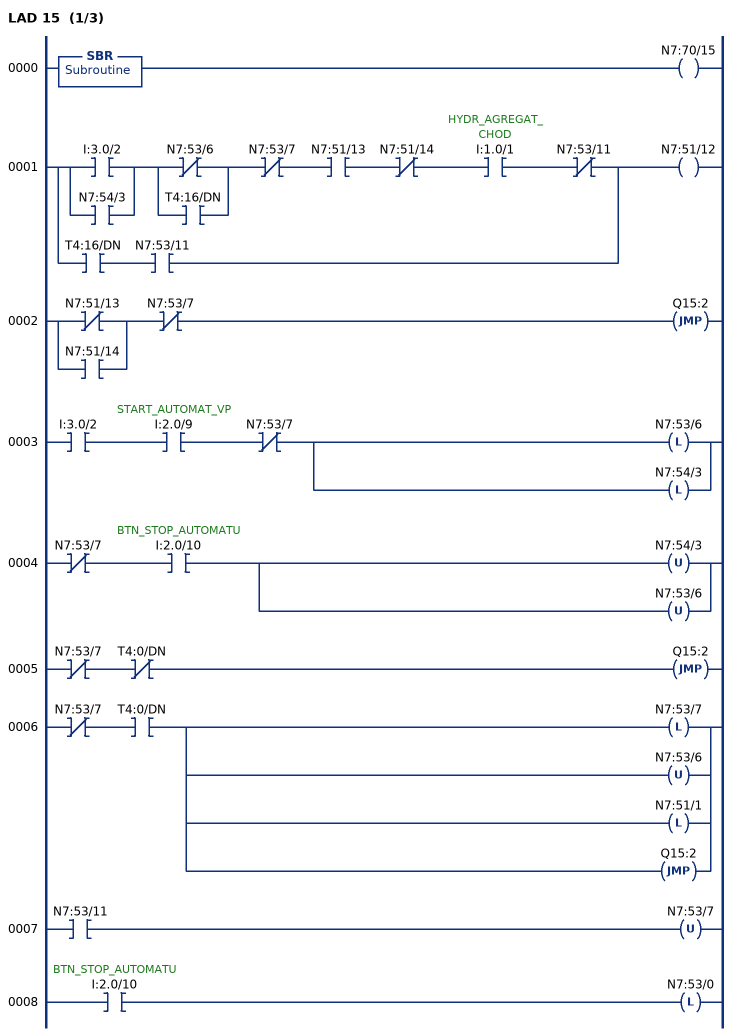
% Rung: 0 %
SOR SBR OTE N7:70/15 EOR
% Rung: 1 %
SOR BST BST XIC I:3.0/2 NXB XIC N7:54/3 BND BST XIO N7:53/6 NXB XIC T4:16/DN BND XIO N7:53/7 XIC N7:51/13 XIO N7:51/14 XIC I:1.0/1 XIO N7:53/11 NXB XIC T4:16/DN XIC N7:53/11 BND OTE N7:51/12 EOR
%   I:1.0/1  HYDR_AGREGAT_CHOD %
% Rung: 2 %
SOR BST XIO N7:51/13 NXB XIC N7:51/14 BND XIO N7:53/7 JMP Q15:2 EOR
% Rung: 3 %
SOR XIC I:3.0/2 XIC I:2.0/9 XIO N7:53/7 BST OTL N7:53/6 NXB OTL N7:54/3 BND EOR
%   I:2.0/9  START_AUTOMAT_VP %
% Rung: 4 %
SOR XIO N7:53/7 XIC I:2.0/10 BST OTU N7:54/3 NXB OTU N7:53/6 BND EOR
%   I:2.0/10  BTN_STOP_AUTOMATU %
% Rung: 5 %
SOR XIO N7:53/7 XIO T4:0/DN JMP Q15:2 EOR
% Rung: 6 %
SOR XIO N7:53/7 XIC T4:0/DN BST OTL N7:53/7 NXB OTU N7:53/6 NXB OTL N7:51/1 NXB JMP Q15:2 BND EOR
% Rung: 7 %
SOR XIC N7:53/11 OTU N7:53/7 EOR
% Rung: 8 %
SOR XIC I:2.0/10 OTL N7:53/0 EOR
%   I:2.0/10  BTN_STOP_AUTOMATU %

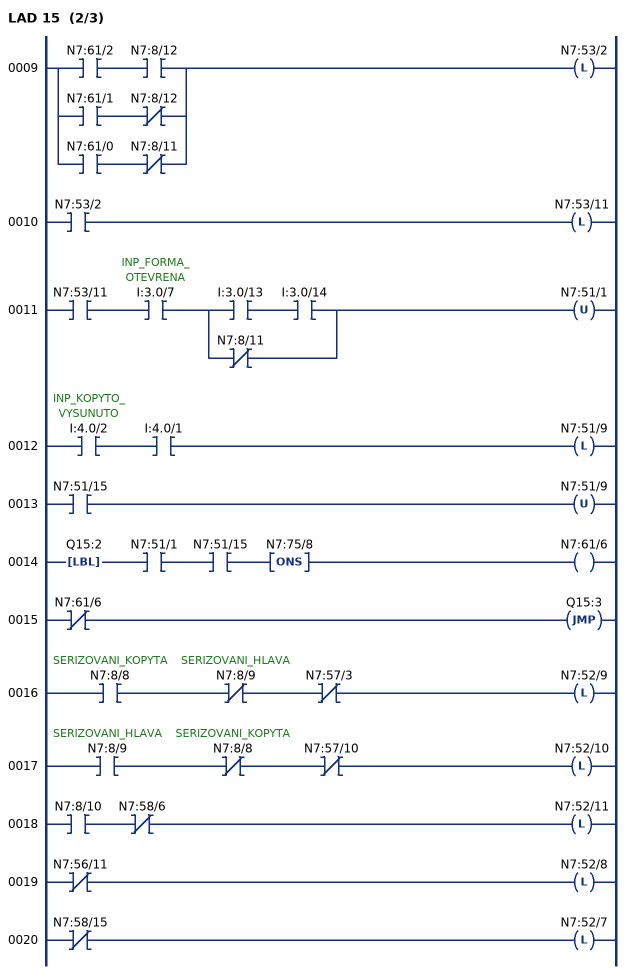
% Rung: 9 %
SOR BST XIC N7:61/2 XIC N7:8/12 NXB XIC N7:61/1 XIO N7:8/12 NXB XIC N7:61/0 XIO N7:8/11 BND OTL N7:53/2 EOR
% Rung: 10 %
SOR XIC N7:53/2 OTL N7:53/11 EOR
% Rung: 11 %
SOR XIC N7:53/11 XIC I:3.0/7 BST XIC I:3.0/13 XIC I:3.0/14 NXB XIO N7:8/11 BND OTU N7:51/1 EOR
%   I:3.0/7  INP_FORMA_OTEVRENA %
% Rung: 12 %
SOR XIC I:4.0/2 XIC I:4.0/1 OTL N7:51/9 EOR
%   I:4.0/2  INP_KOPYTO_VYSUNUTO %
% Rung: 13 %
SOR XIC N7:51/15 OTU N7:51/9 EOR
% Rung: 14 %
SOR LBL Q15:2 XIC N7:51/1 XIC N7:51/15 OSR N7:75/8 OTE N7:61/6 EOR
% Rung: 15 %
SOR XIO N7:61/6 JMP Q15:3 EOR
% Rung: 16 %
SOR XIC N7:8/8 XIO N7:8/9 XIO N7:57/3 OTL N7:52/9 EOR
%   N7:8/8  SERIZOVANI_KOPYTA %
%   N7:8/9  SERIZOVANI_HLAVA %
% Rung: 17 %
SOR XIC N7:8/9 XIO N7:8/8 XIO N7:57/10 OTL N7:52/10 EOR
%   N7:8/9  SERIZOVANI_HLAVA %
%   N7:8/8  SERIZOVANI_KOPYTA %
% Rung: 18 %
SOR XIC N7:8/10 XIO N7:58/6 OTL N7:52/11 EOR
% Rung: 19 %
SOR XIO N7:56/11 OTL N7:52/8 EOR
% Rung: 20 %
SOR XIO N7:58/15 OTL N7:52/7 EOR

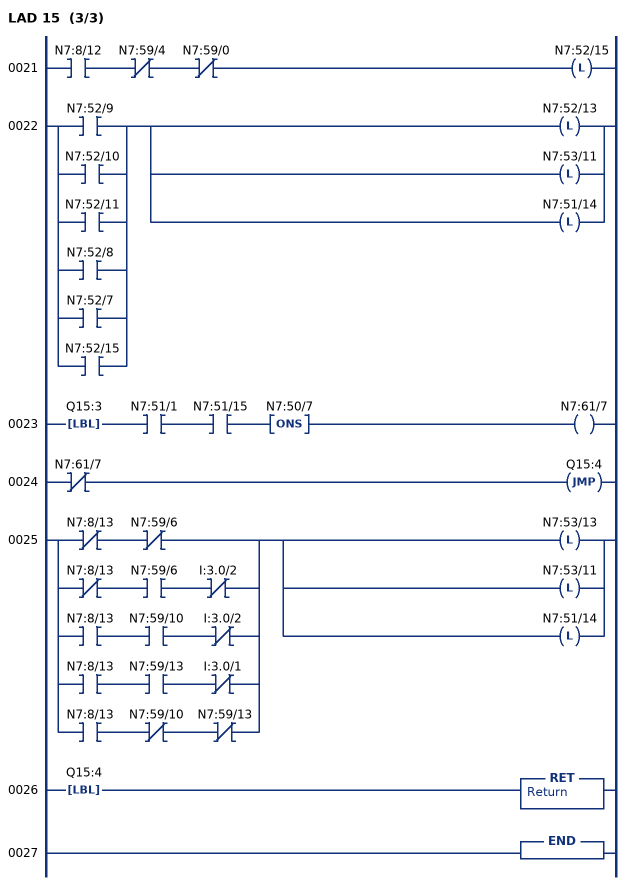
% Rung: 21 %
SOR XIC N7:8/12 XIO N7:59/4 XIO N7:59/0 OTL N7:52/15 EOR
% Rung: 22 %
SOR BST XIC N7:52/9 NXB XIC N7:52/10 NXB XIC N7:52/11 NXB XIC N7:52/8 NXB XIC N7:52/7 NXB XIC N7:52/15 BND BST OTL N7:52/13 NXB OTL N7:53/11 NXB OTL N7:51/14 BND EOR
% Rung: 23 %
SOR LBL Q15:3 XIC N7:51/1 XIC N7:51/15 OSR N7:50/7 OTE N7:61/7 EOR
% Rung: 24 %
SOR XIO N7:61/7 JMP Q15:4 EOR
% Rung: 25 %
SOR BST XIO N7:8/13 XIO N7:59/6 NXB XIO N7:8/13 XIC N7:59/6 XIO I:3.0/2 NXB XIC N7:8/13 XIC N7:59/10 XIO I:3.0/2 NXB XIC N7:8/13 XIC N7:59/13 XIO I:3.0/1 NXB XIC N7:8/13 XIO N7:59/10 XIO N7:59/13 BND BST OTL N7:53/13 NXB OTL N7:53/11 NXB OTL N7:51/14 BND EOR
% Rung: 26 %
SOR LBL Q15:4 RET EOR
% Rung: 27 %
SOR END EOR

LADDER 16
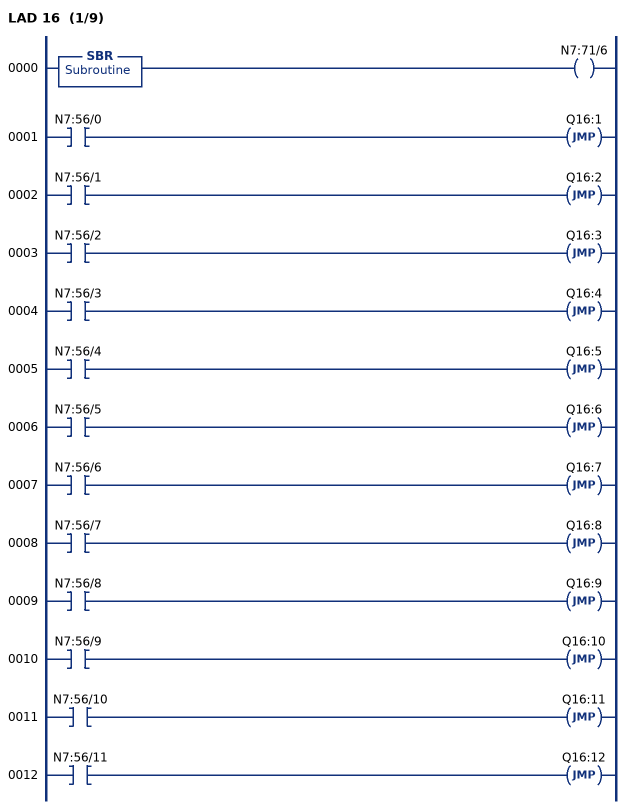
% Rung: 0 %
SOR SBR OTE N7:71/6 EOR
% Rung: 1 %
SOR XIC N7:56/0 JMP Q16:1 EOR
% Rung: 2 %
SOR XIC N7:56/1 JMP Q16:2 EOR
% Rung: 3 %
SOR XIC N7:56/2 JMP Q16:3 EOR
% Rung: 4 %
SOR XIC N7:56/3 JMP Q16:4 EOR
% Rung: 5 %
SOR XIC N7:56/4 JMP Q16:5 EOR
% Rung: 6 %
SOR XIC N7:56/5 JMP Q16:6 EOR
% Rung: 7 %
SOR XIC N7:56/6 JMP Q16:7 EOR
% Rung: 8 %
SOR XIC N7:56/7 JMP Q16:8 EOR
% Rung: 9 %
SOR XIC N7:56/8 JMP Q16:9 EOR
% Rung: 10 %
SOR XIC N7:56/9 JMP Q16:10 EOR
% Rung: 11 %
SOR XIC N7:56/10 JMP Q16:11 EOR
% Rung: 12 %
SOR XIC N7:56/11 JMP Q16:12 EOR

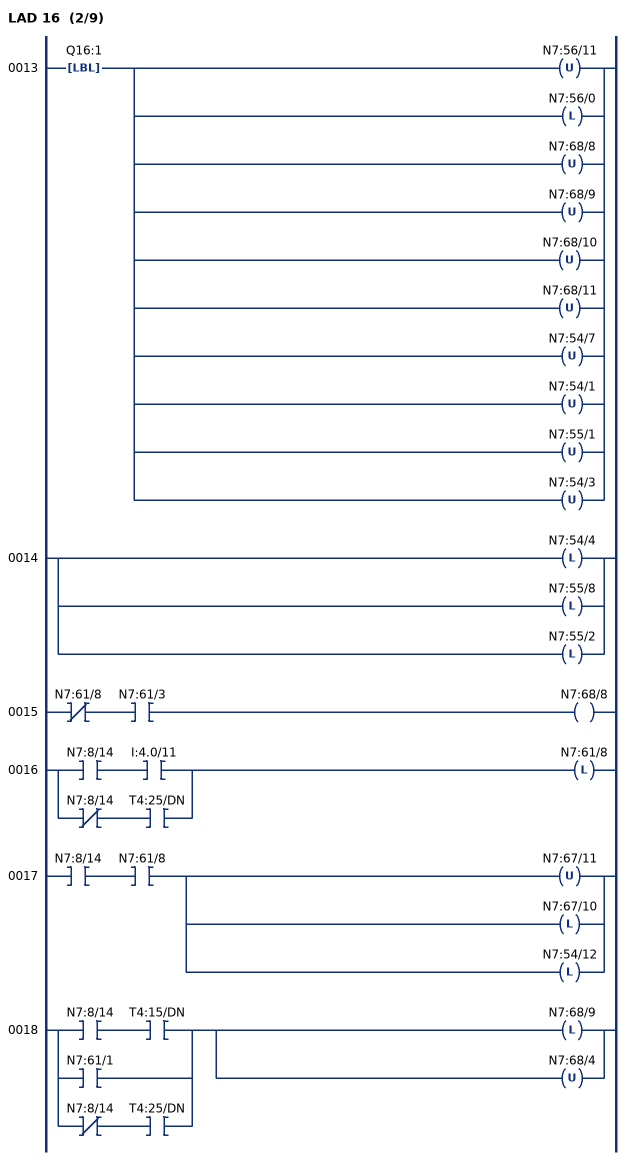
% Rung: 13 %
SOR LBL Q16:1 BST BST OTU N7:56/11 NXB OTL N7:56/0 BND NXB OTU N7:68/8 NXB OTU N7:68/9 NXB OTU N7:68/10 NXB OTU N7:68/11 NXB OTU N7:54/7 NXB OTU N7:54/1 NXB OTU N7:55/1 NXB OTU N7:54/3 BND EOR
% Rung: 14 %
SOR BST OTL N7:54/4 NXB OTL N7:55/8 NXB OTL N7:55/2 BND EOR
% Rung: 15 %
SOR XIO N7:61/8 XIC N7:61/3 OTE N7:68/8 EOR
% Rung: 16 %
SOR BST XIC N7:8/14 XIC I:4.0/11 NXB XIO N7:8/14 XIC T4:25/DN BND OTL N7:61/8 EOR
% Rung: 17 %
SOR XIC N7:8/14 XIC N7:61/8 BST OTU N7:67/11 NXB OTL N7:67/10 NXB OTL N7:54/12 BND EOR
% Rung: 18 %
SOR BST XIC N7:8/14 XIC T4:15/DN NXB XIC N7:61/1 NXB XIO N7:8/14 XIC T4:25/DN BND BST OTL N7:68/9 NXB OTU N7:68/4 BND EOR

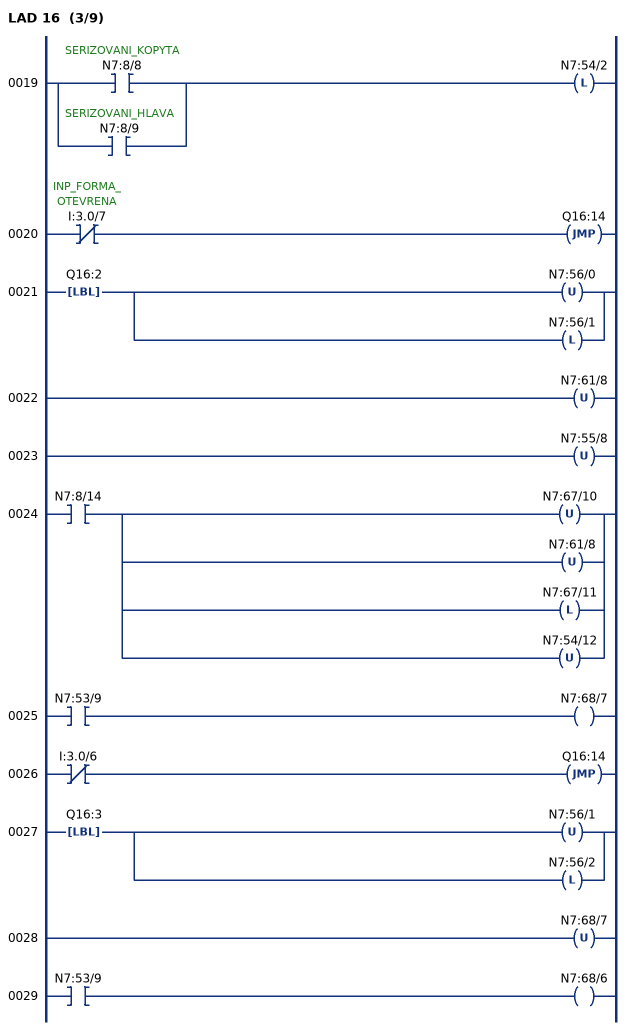
% Rung: 19 %
SOR BST XIC N7:8/8 NXB XIC N7:8/9 BND OTL N7:54/2 EOR
%   N7:8/8  SERIZOVANI_KOPYTA %
%   N7:8/9  SERIZOVANI_HLAVA %
% Rung: 20 %
SOR XIO I:3.0/7 JMP Q16:14 EOR
%   I:3.0/7  INP_FORMA_OTEVRENA %
% Rung: 21 %
SOR LBL Q16:2 BST OTU N7:56/0 NXB OTL N7:56/1 BND EOR
% Rung: 22 %
SOR OTU N7:61/8 EOR
% Rung: 23 %
SOR OTU N7:55/8 EOR
% Rung: 24 %
SOR XIC N7:8/14 BST OTU N7:67/10 NXB OTU N7:61/8 NXB OTL N7:67/11 NXB OTU N7:54/12 BND EOR
% Rung: 25 %
SOR XIC N7:53/9 OTE N7:68/7 EOR
% Rung: 26 %
SOR XIO I:3.0/6 JMP Q16:14 EOR
% Rung: 27 %
SOR LBL Q16:3 BST OTU N7:56/1 NXB OTL N7:56/2 BND EOR
% Rung: 28 %
SOR OTU N7:68/7 EOR
% Rung: 29 %
SOR XIC N7:53/9 OTE N7:68/6 EOR

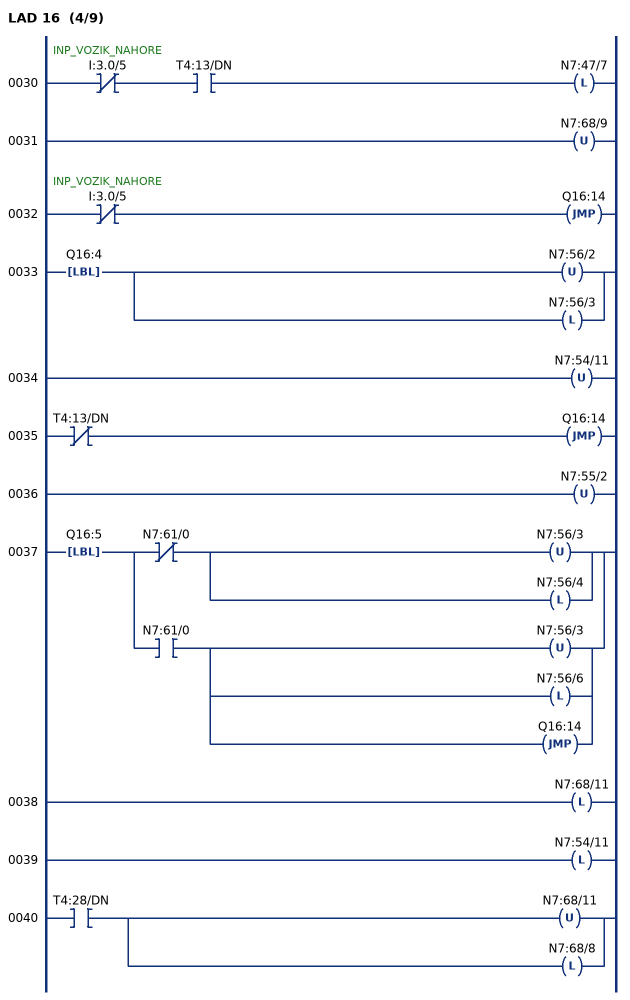
% Rung: 30 %
SOR XIO I:3.0/5 XIC T4:13/DN OTL N7:47/7 EOR
%   I:3.0/5  INP_VOZIK_NAHORE %
% Rung: 31 %
SOR OTU N7:68/9 EOR
% Rung: 32 %
SOR XIO I:3.0/5 JMP Q16:14 EOR
%   I:3.0/5  INP_VOZIK_NAHORE %
% Rung: 33 %
SOR LBL Q16:4 BST OTU N7:56/2 NXB OTL N7:56/3 BND EOR
% Rung: 34 %
SOR OTU N7:54/11 EOR
% Rung: 35 %
SOR XIO T4:13/DN JMP Q16:14 EOR
% Rung: 36 %
SOR OTU N7:55/2 EOR
% Rung: 37 %
SOR LBL Q16:5 BST XIO N7:61/0 BST OTU N7:56/3 NXB OTL N7:56/4 BND NXB XIC N7:61/0 BST OTU N7:56/3 NXB OTL N7:56/6 NXB JMP Q16:14 BND BND EOR
% Rung: 38 %
SOR OTL N7:68/11 EOR
% Rung: 39 %
SOR OTL N7:54/11 EOR
% Rung: 40 %
SOR XIC T4:28/DN BST OTU N7:68/11 NXB OTL N7:68/8 BND EOR

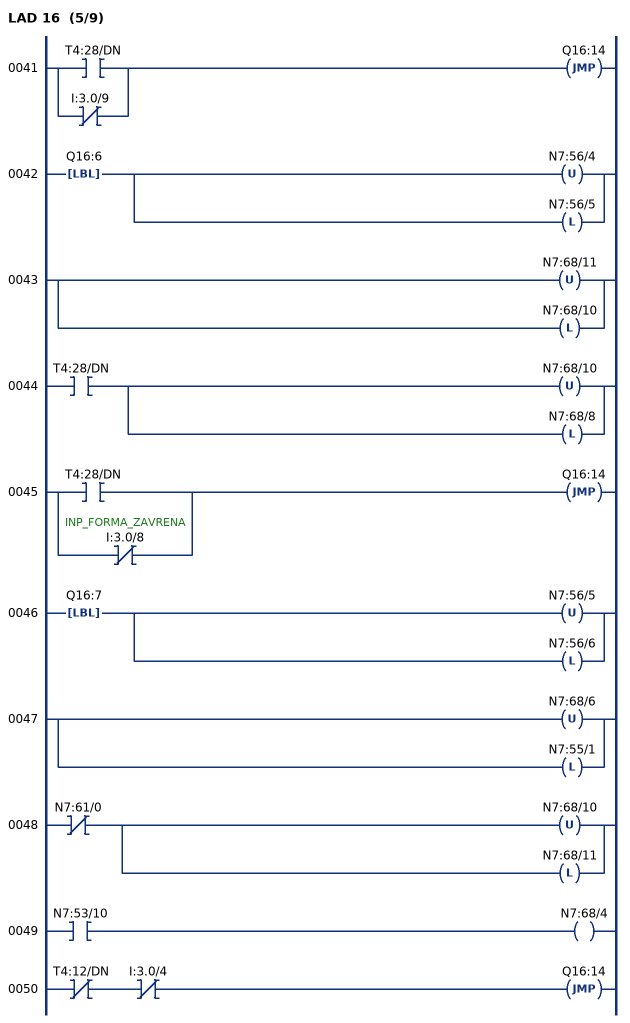
% Rung: 41 %
SOR BST XIC T4:28/DN NXB XIO I:3.0/9 BND JMP Q16:14 EOR
% Rung: 42 %
SOR LBL Q16:6 BST OTU N7:56/4 NXB OTL N7:56/5 BND EOR
% Rung: 43 %
SOR BST OTU N7:68/11 NXB OTL N7:68/10 BND EOR
% Rung: 44 %
SOR XIC T4:28/DN BST OTU N7:68/10 NXB OTL N7:68/8 BND EOR
% Rung: 45 %
SOR BST XIC T4:28/DN NXB XIO I:3.0/8 BND JMP Q16:14 EOR
%   I:3.0/8  INP_FORMA_ZAVRENA %
% Rung: 46 %
SOR LBL Q16:7 BST OTU N7:56/5 NXB OTL N7:56/6 BND EOR
% Rung: 47 %
SOR BST OTU N7:68/6 NXB OTL N7:55/1 BND EOR
% Rung: 48 %
SOR XIO N7:61/0 BST OTU N7:68/10 NXB OTL N7:68/11 BND EOR
% Rung: 49 %
SOR XIC N7:53/10 OTE N7:68/4 EOR
% Rung: 50 %
SOR XIO T4:12/DN XIO I:3.0/4 JMP Q16:14 EOR

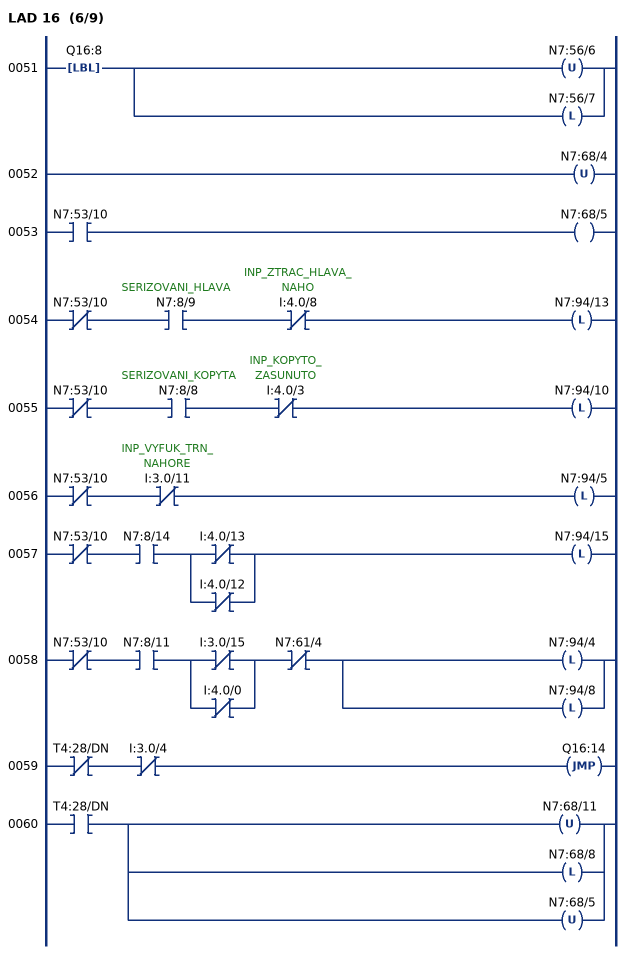
% Rung: 51 %
SOR LBL Q16:8 BST OTU N7:56/6 NXB OTL N7:56/7 BND EOR
% Rung: 52 %
SOR OTU N7:68/4 EOR
% Rung: 53 %
SOR XIC N7:53/10 OTE N7:68/5 EOR
% Rung: 54 %
SOR XIO N7:53/10 XIC N7:8/9 XIO I:4.0/8 OTL N7:94/13 EOR
%   N7:8/9  SERIZOVANI_HLAVA %
%   I:4.0/8  INP_ZTRAC_HLAVA_NAHO %
% Rung: 55 %
SOR XIO N7:53/10 XIC N7:8/8 XIO I:4.0/3 OTL N7:94/10 EOR
%   N7:8/8  SERIZOVANI_KOPYTA %
%   I:4.0/3  INP_KOPYTO_ZASUNUTO %
% Rung: 56 %
SOR XIO N7:53/10 XIO I:3.0/11 OTL N7:94/5 EOR
%   I:3.0/11  INP_VYFUK_TRN_NAHORE %
% Rung: 57 %
SOR XIO N7:53/10 XIC N7:8/14 BST XIO I:4.0/13 NXB XIO I:4.0/12 BND OTL N7:94/15 EOR
% Rung: 58 %
SOR XIO N7:53/10 XIC N7:8/11 BST XIO I:3.0/15 NXB XIO I:4.0/0 BND XIO N7:61/4 BST OTL N7:94/4 NXB OTL N7:94/8 BND EOR
% Rung: 59 %
SOR XIO T4:28/DN XIO I:3.0/4 JMP Q16:14 EOR
% Rung: 60 %
SOR XIC T4:28/DN BST OTU N7:68/11 NXB OTL N7:68/8 NXB OTU N7:68/5 BND EOR

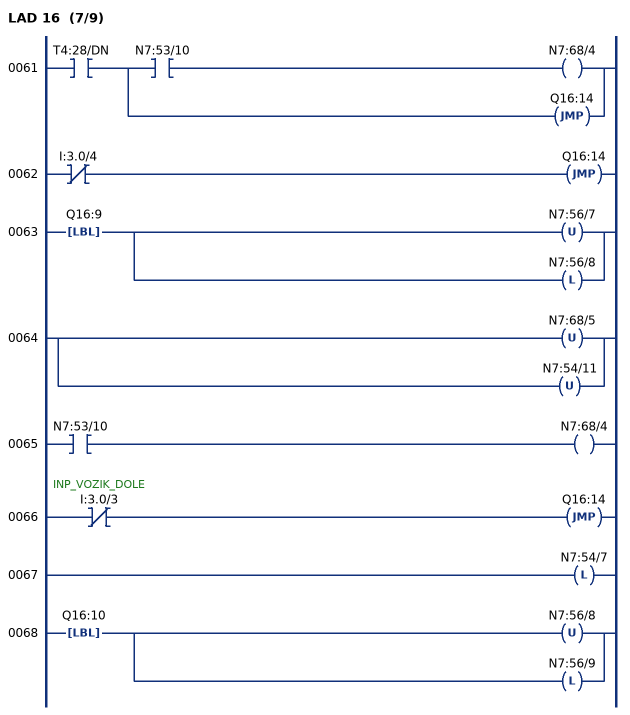
% Rung: 61 %
SOR XIC T4:28/DN BST XIC N7:53/10 OTE N7:68/4 NXB JMP Q16:14 BND EOR
% Rung: 62 %
SOR XIO I:3.0/4 JMP Q16:14 EOR
% Rung: 63 %
SOR LBL Q16:9 BST OTU N7:56/7 NXB OTL N7:56/8 BND EOR
% Rung: 64 %
SOR BST OTU N7:68/5 NXB OTU N7:54/11 BND EOR
% Rung: 65 %
SOR XIC N7:53/10 OTE N7:68/4 EOR
% Rung: 66 %
SOR XIO I:3.0/3 JMP Q16:14 EOR
%   I:3.0/3  INP_VOZIK_DOLE %
% Rung: 67 %
SOR OTL N7:54/7 EOR
% Rung: 68 %
SOR LBL Q16:10 BST OTU N7:56/8 NXB OTL N7:56/9 BND EOR

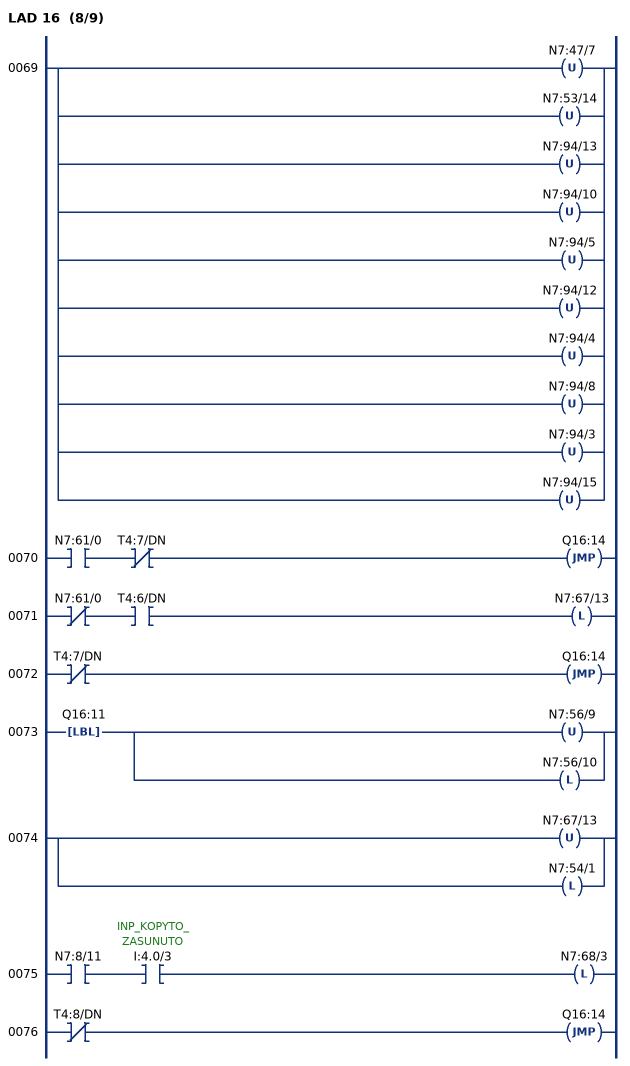
% Rung: 69 %
SOR BST OTU N7:47/7 NXB OTU N7:53/14 NXB OTU N7:94/13 NXB OTU N7:94/10 NXB OTU N7:94/5 NXB OTU N7:94/12 NXB OTU N7:94/4 NXB OTU N7:94/8 NXB OTU N7:94/3 NXB OTU N7:94/15 BND EOR
% Rung: 70 %
SOR XIC N7:61/0 XIO T4:7/DN JMP Q16:14 EOR
% Rung: 71 %
SOR XIO N7:61/0 XIC T4:6/DN OTL N7:67/13 EOR
% Rung: 72 %
SOR XIO T4:7/DN JMP Q16:14 EOR
% Rung: 73 %
SOR LBL Q16:11 BST OTU N7:56/9 NXB OTL N7:56/10 BND EOR
% Rung: 74 %
SOR BST OTU N7:67/13 NXB OTL N7:54/1 BND EOR
% Rung: 75 %
SOR XIC N7:8/11 XIC I:4.0/3 OTL N7:68/3 EOR
%   I:4.0/3  INP_KOPYTO_ZASUNUTO %
% Rung: 76 %
SOR XIO T4:8/DN JMP Q16:14 EOR

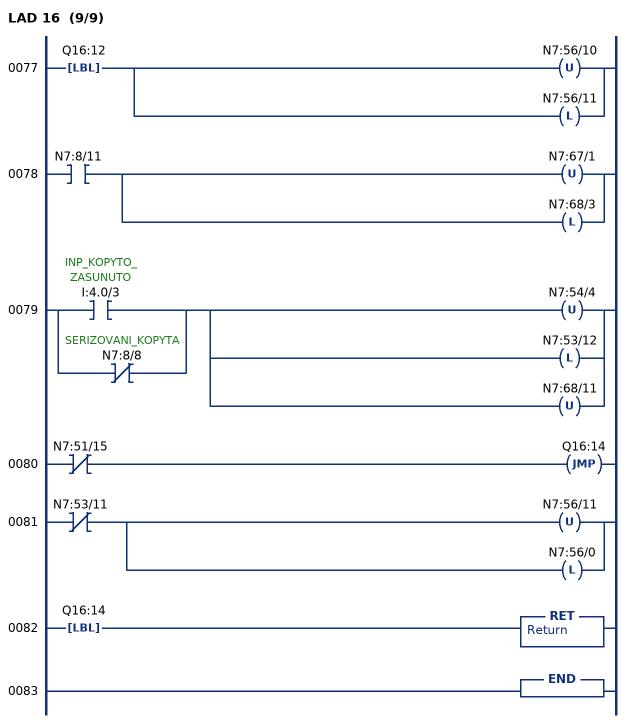
% Rung: 77 %
SOR LBL Q16:12 BST OTU N7:56/10 NXB OTL N7:56/11 BND EOR
% Rung: 78 %
SOR XIC N7:8/11 BST OTU N7:67/1 NXB OTL N7:68/3 BND EOR
% Rung: 79 %
SOR BST XIC I:4.0/3 NXB XIO N7:8/8 BND BST OTU N7:54/4 NXB OTL N7:53/12 NXB OTU N7:68/11 BND EOR
%   I:4.0/3  INP_KOPYTO_ZASUNUTO %
%   N7:8/8  SERIZOVANI_KOPYTA %
% Rung: 80 %
SOR XIO N7:51/15 JMP Q16:14 EOR
% Rung: 81 %
SOR XIO N7:53/11 BST OTU N7:56/11 NXB OTL N7:56/0 BND EOR
% Rung: 82 %
SOR LBL Q16:14 RET EOR
% Rung: 83 %
SOR END EOR

LADDER 17
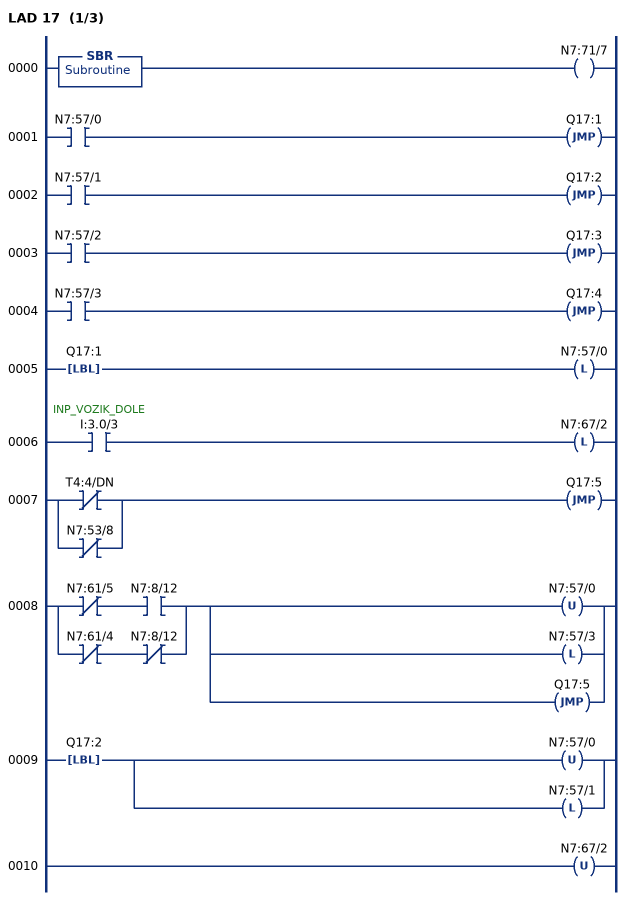
% Rung: 0 %
SOR SBR OTE N7:71/7 EOR
% Rung: 1 %
SOR XIC N7:57/0 JMP Q17:1 EOR
% Rung: 2 %
SOR XIC N7:57/1 JMP Q17:2 EOR
% Rung: 3 %
SOR XIC N7:57/2 JMP Q17:3 EOR
% Rung: 4 %
SOR XIC N7:57/3 JMP Q17:4 EOR
% Rung: 5 %
SOR LBL Q17:1 OTL N7:57/0 EOR
% Rung: 6 %
SOR XIC I:3.0/3 OTL N7:67/2 EOR
%   I:3.0/3  INP_VOZIK_DOLE %
% Rung: 7 %
SOR BST XIO T4:4/DN NXB XIO N7:53/8 BND JMP Q17:5 EOR
% Rung: 8 %
SOR BST XIO N7:61/5 XIC N7:8/12 NXB XIO N7:61/4 XIO N7:8/12 BND BST OTU N7:57/0 NXB OTL N7:57/3 NXB JMP Q17:5 BND EOR
% Rung: 9 %
SOR LBL Q17:2 BST OTU N7:57/0 NXB OTL N7:57/1 BND EOR
% Rung: 10 %
SOR OTU N7:67/2 EOR

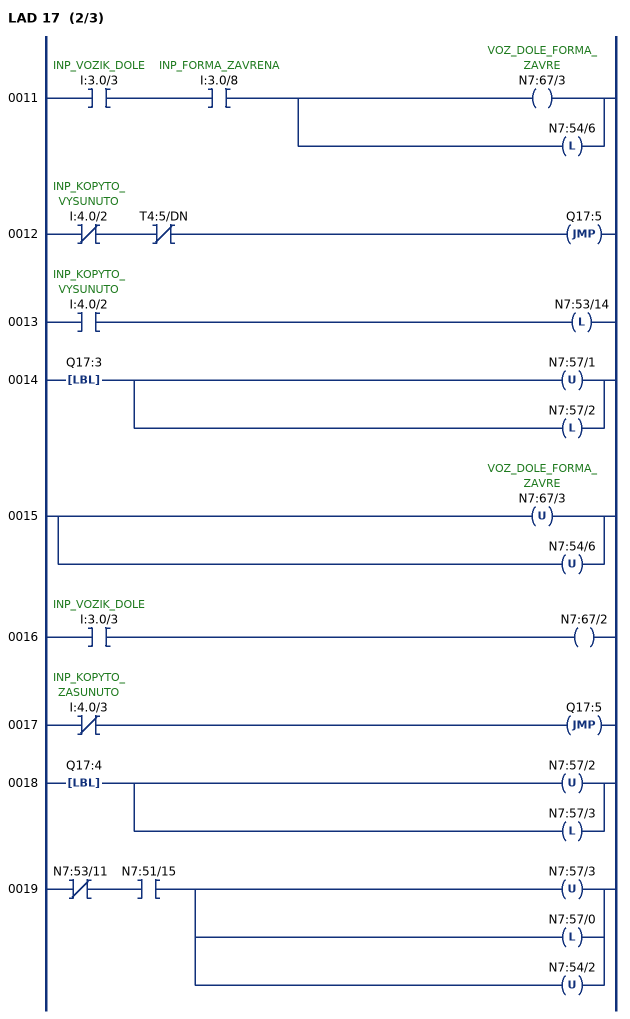
% Rung: 11 %
SOR XIC I:3.0/3 XIC I:3.0/8 BST OTE N7:67/3 NXB OTL N7:54/6 BND EOR
%   I:3.0/3  INP_VOZIK_DOLE %
%   I:3.0/8  INP_FORMA_ZAVRENA %
%   N7:67/3  VOZ_DOLE_FORMA_ZAVRE %
% Rung: 12 %
SOR XIO I:4.0/2 XIO T4:5/DN JMP Q17:5 EOR
%   I:4.0/2  INP_KOPYTO_VYSUNUTO %
% Rung: 13 %
SOR XIC I:4.0/2 OTL N7:53/14 EOR
%   I:4.0/2  INP_KOPYTO_VYSUNUTO %
% Rung: 14 %
SOR LBL Q17:3 BST OTU N7:57/1 NXB OTL N7:57/2 BND EOR
% Rung: 15 %
SOR BST OTU N7:67/3 NXB OTU N7:54/6 BND EOR
%   N7:67/3  VOZ_DOLE_FORMA_ZAVRE %
% Rung: 16 %
SOR XIC I:3.0/3 OTE N7:67/2 EOR
%   I:3.0/3  INP_VOZIK_DOLE %
% Rung: 17 %
SOR XIO I:4.0/3 JMP Q17:5 EOR
%   I:4.0/3  INP_KOPYTO_ZASUNUTO %
% Rung: 18 %
SOR LBL Q17:4 BST OTU N7:57/2 NXB OTL N7:57/3 BND EOR
% Rung: 19 %
SOR XIO N7:53/11 XIC N7:51/15 BST OTU N7:57/3 NXB OTL N7:57/0 NXB OTU N7:54/2 BND EOR

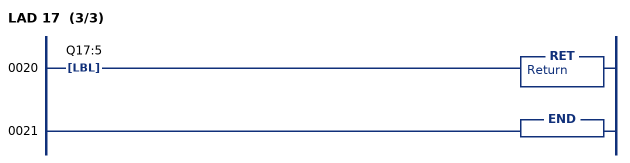
% Rung: 20 %
SOR LBL Q17:5 RET EOR
% Rung: 21 %
SOR END EOR

LADDER 18
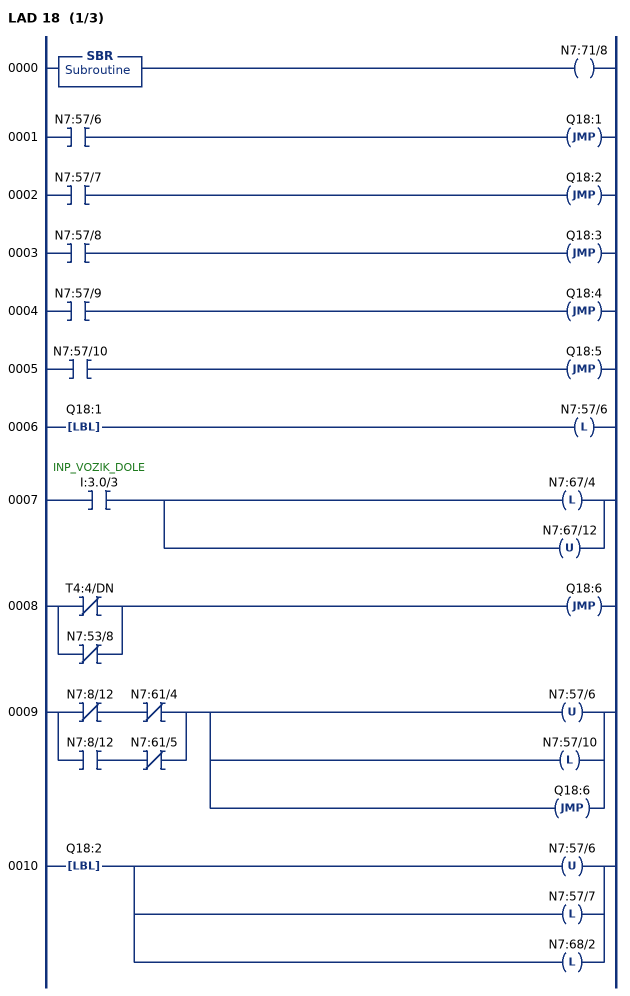
% Rung: 0 %
SOR SBR OTE N7:71/8 EOR
% Rung: 1 %
SOR XIC N7:57/6 JMP Q18:1 EOR
% Rung: 2 %
SOR XIC N7:57/7 JMP Q18:2 EOR
% Rung: 3 %
SOR XIC N7:57/8 JMP Q18:3 EOR
% Rung: 4 %
SOR XIC N7:57/9 JMP Q18:4 EOR
% Rung: 5 %
SOR XIC N7:57/10 JMP Q18:5 EOR
% Rung: 6 %
SOR LBL Q18:1 OTL N7:57/6 EOR
% Rung: 7 %
SOR XIC I:3.0/3 BST OTL N7:67/4 NXB OTU N7:67/12 BND EOR
%   I:3.0/3  INP_VOZIK_DOLE %
% Rung: 8 %
SOR BST XIO T4:4/DN NXB XIO N7:53/8 BND JMP Q18:6 EOR
% Rung: 9 %
SOR BST XIO N7:8/12 XIO N7:61/4 NXB XIC N7:8/12 XIO N7:61/5 BND BST OTU N7:57/6 NXB BST OTL N7:57/10 NXB JMP Q18:6 BND BND EOR
% Rung: 10 %
SOR LBL Q18:2 BST OTU N7:57/6 NXB OTL N7:57/7 NXB OTL N7:68/2 BND EOR

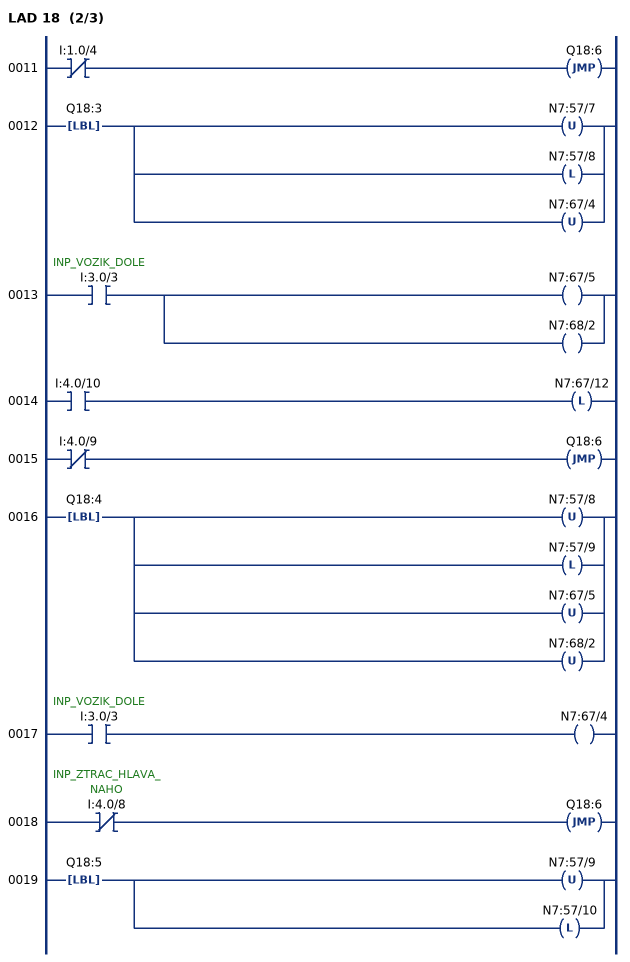
% Rung: 11 %
SOR XIO I:1.0/4 JMP Q18:6 EOR
% Rung: 12 %
SOR LBL Q18:3 BST OTU N7:57/7 NXB OTL N7:57/8 NXB OTU N7:67/4 BND EOR
% Rung: 13 %
SOR XIC I:3.0/3 BST OTE N7:67/5 NXB OTE N7:68/2 BND EOR
%   I:3.0/3  INP_VOZIK_DOLE %
% Rung: 14 %
SOR XIC I:4.0/10 OTL N7:67/12 EOR
% Rung: 15 %
SOR XIO I:4.0/9 JMP Q18:6 EOR
% Rung: 16 %
SOR LBL Q18:4 BST OTU N7:57/8 NXB OTL N7:57/9 NXB OTU N7:67/5 NXB OTU N7:68/2 BND EOR
% Rung: 17 %
SOR XIC I:3.0/3 OTE N7:67/4 EOR
%   I:3.0/3  INP_VOZIK_DOLE %
% Rung: 18 %
SOR XIO I:4.0/8 JMP Q18:6 EOR
%   I:4.0/8  INP_ZTRAC_HLAVA_NAHO %
% Rung: 19 %
SOR LBL Q18:5 BST OTU N7:57/9 NXB OTL N7:57/10 BND EOR

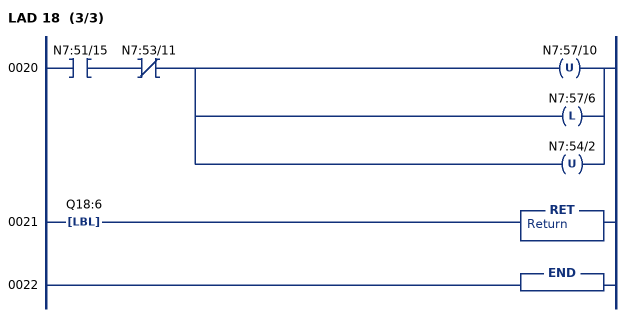
% Rung: 20 %
SOR XIC N7:51/15 XIO N7:53/11 BST OTU N7:57/10 NXB OTL N7:57/6 NXB OTU N7:54/2 BND EOR
% Rung: 21 %
SOR LBL Q18:6 RET EOR
% Rung: 22 %
SOR END EOR

LADDER 19
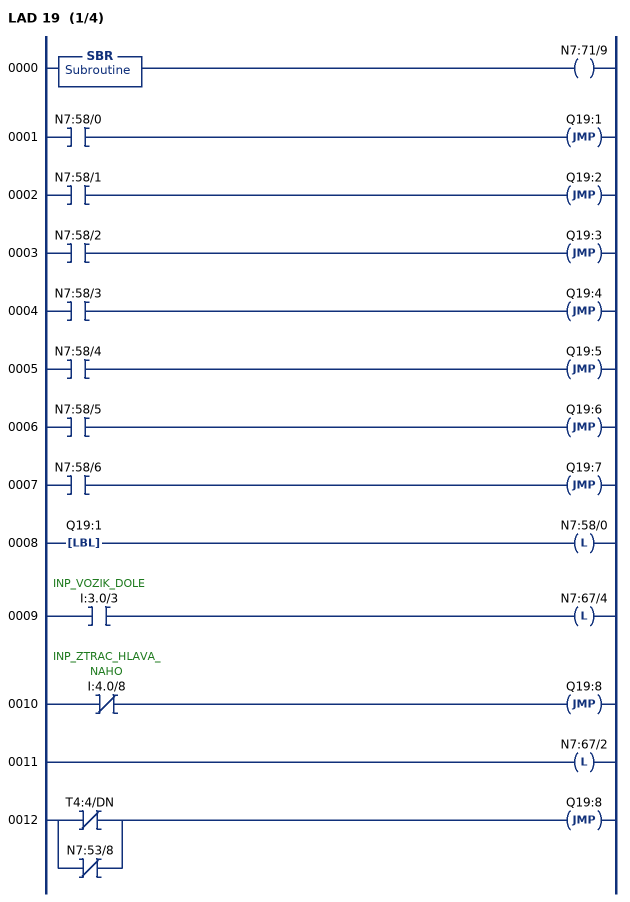
% Rung: 0 %
SOR SBR OTE N7:71/9 EOR
% Rung: 1 %
SOR XIC N7:58/0 JMP Q19:1 EOR
% Rung: 2 %
SOR XIC N7:58/1 JMP Q19:2 EOR
% Rung: 3 %
SOR XIC N7:58/2 JMP Q19:3 EOR
% Rung: 4 %
SOR XIC N7:58/3 JMP Q19:4 EOR
% Rung: 5 %
SOR XIC N7:58/4 JMP Q19:5 EOR
% Rung: 6 %
SOR XIC N7:58/5 JMP Q19:6 EOR
% Rung: 7 %
SOR XIC N7:58/6 JMP Q19:7 EOR
% Rung: 8 %
SOR LBL Q19:1 OTL N7:58/0 EOR
% Rung: 9 %
SOR XIC I:3.0/3 OTL N7:67/4 EOR
%   I:3.0/3  INP_VOZIK_DOLE %
% Rung: 10 %
SOR XIO I:4.0/8 JMP Q19:8 EOR
%   I:4.0/8  INP_ZTRAC_HLAVA_NAHO %
% Rung: 11 %
SOR OTL N7:67/2 EOR
% Rung: 12 %
SOR BST XIO T4:4/DN NXB XIO N7:53/8 BND JMP Q19:8 EOR

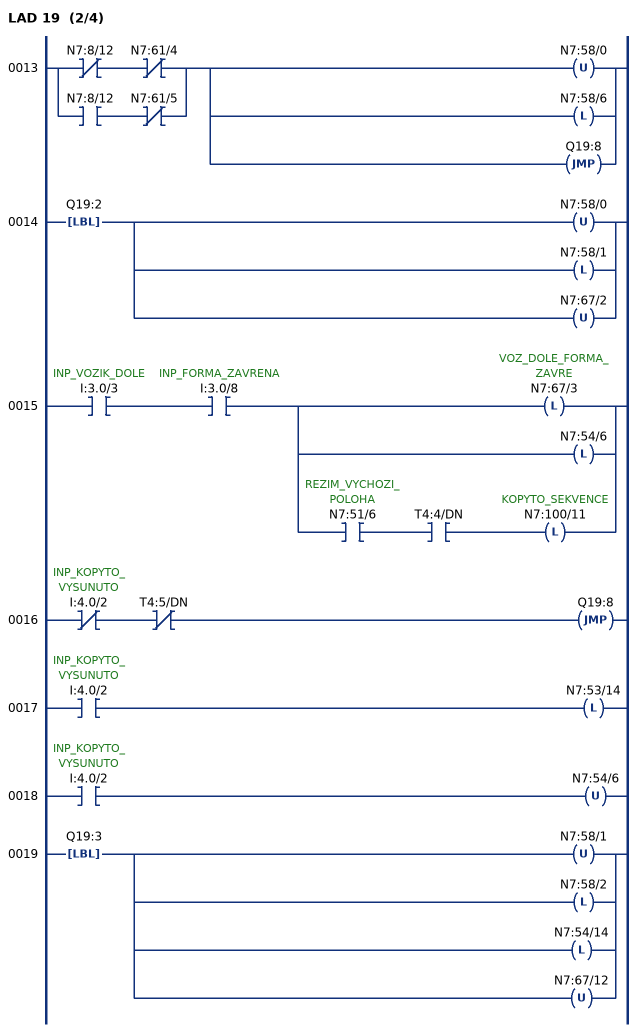
% Rung: 13 %
SOR BST XIO N7:8/12 XIO N7:61/4 NXB XIC N7:8/12 XIO N7:61/5 BND BST OTU N7:58/0 NXB OTL N7:58/6 NXB JMP Q19:8 BND EOR
% Rung: 14 %
SOR LBL Q19:2 BST OTU N7:58/0 NXB OTL N7:58/1 NXB OTU N7:67/2 BND EOR
% Rung: 15 %
SOR XIC I:3.0/3 XIC I:3.0/8 BST OTL N7:67/3 NXB OTL N7:54/6 NXB XIC N7:51/6 XIC T4:4/DN OTL N7:100/11 BND EOR
%   I:3.0/3  INP_VOZIK_DOLE %
%   I:3.0/8  INP_FORMA_ZAVRENA %
%   N7:67/3  VOZ_DOLE_FORMA_ZAVRE %
%   N7:51/6  REZIM_VYCHOZI_POLOHA %
%   N7:100/11  KOPYTO_SEKVENCE %
% Rung: 16 %
SOR XIO I:4.0/2 XIO T4:5/DN JMP Q19:8 EOR
%   I:4.0/2  INP_KOPYTO_VYSUNUTO %
% Rung: 17 %
SOR XIC I:4.0/2 OTL N7:53/14 EOR
%   I:4.0/2  INP_KOPYTO_VYSUNUTO %
% Rung: 18 %
SOR XIC I:4.0/2 OTU N7:54/6 EOR
%   I:4.0/2  INP_KOPYTO_VYSUNUTO %
% Rung: 19 %
SOR LBL Q19:3 BST OTU N7:58/1 NXB OTL N7:58/2 NXB OTL N7:54/14 NXB OTU N7:67/12 BND EOR

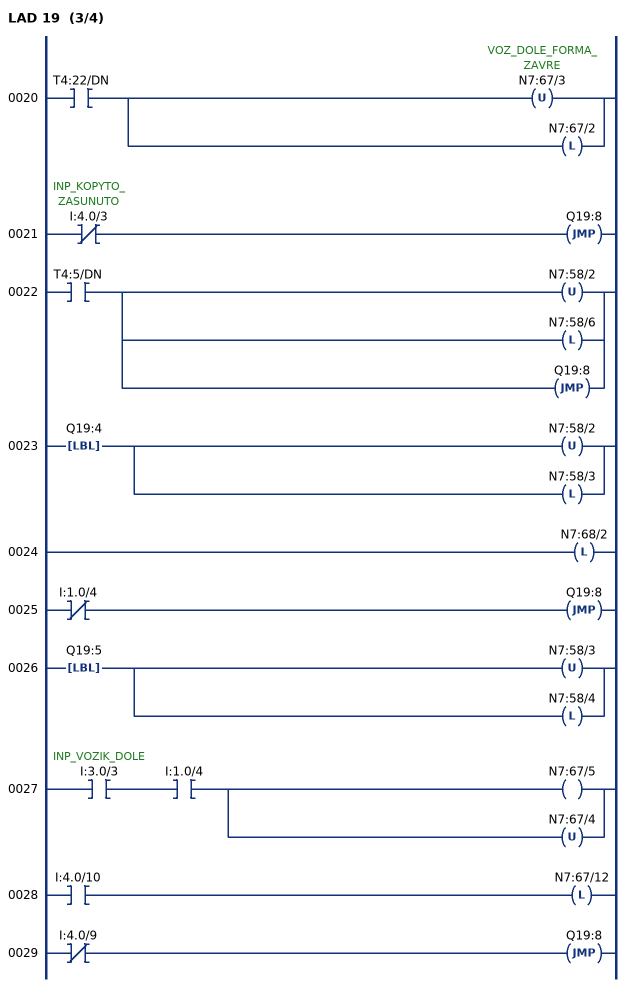
% Rung: 20 %
SOR XIC T4:22/DN BST OTU N7:67/3 NXB OTL N7:67/2 BND EOR
%   N7:67/3  VOZ_DOLE_FORMA_ZAVRE %
% Rung: 21 %
SOR XIO I:4.0/3 JMP Q19:8 EOR
%   I:4.0/3  INP_KOPYTO_ZASUNUTO %
% Rung: 22 %
SOR XIC T4:5/DN BST OTU N7:58/2 NXB OTL N7:58/6 NXB JMP Q19:8 BND EOR
% Rung: 23 %
SOR LBL Q19:4 BST OTU N7:58/2 NXB OTL N7:58/3 BND EOR
% Rung: 24 %
SOR OTL N7:68/2 EOR
% Rung: 25 %
SOR XIO I:1.0/4 JMP Q19:8 EOR
% Rung: 26 %
SOR LBL Q19:5 BST OTU N7:58/3 NXB OTL N7:58/4 BND EOR
% Rung: 27 %
SOR XIC I:3.0/3 XIC I:1.0/4 BST OTE N7:67/5 NXB OTU N7:67/4 BND EOR
%   I:3.0/3  INP_VOZIK_DOLE %
% Rung: 28 %
SOR XIC I:4.0/10 OTL N7:67/12 EOR
% Rung: 29 %
SOR XIO I:4.0/9 JMP Q19:8 EOR

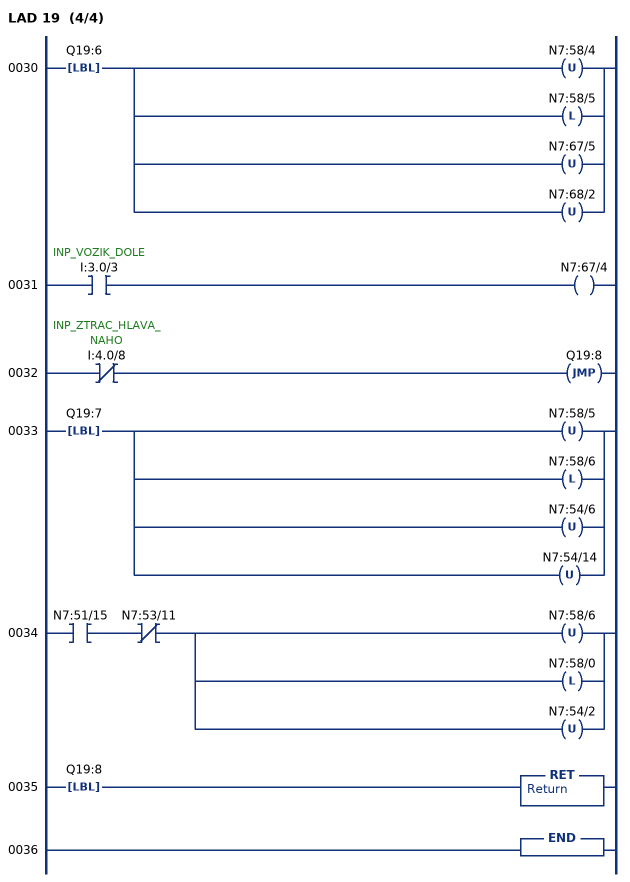
% Rung: 30 %
SOR LBL Q19:6 BST OTU N7:58/4 NXB OTL N7:58/5 NXB OTU N7:67/5 NXB OTU N7:68/2 BND EOR
% Rung: 31 %
SOR XIC I:3.0/3 OTE N7:67/4 EOR
%   I:3.0/3  INP_VOZIK_DOLE %
% Rung: 32 %
SOR XIO I:4.0/8 JMP Q19:8 EOR
%   I:4.0/8  INP_ZTRAC_HLAVA_NAHO %
% Rung: 33 %
SOR LBL Q19:7 BST OTU N7:58/5 NXB OTL N7:58/6 NXB OTU N7:54/6 NXB OTU N7:54/14 BND EOR
% Rung: 34 %
SOR XIC N7:51/15 XIO N7:53/11 BST OTU N7:58/6 NXB OTL N7:58/0 NXB OTU N7:54/2 BND EOR
% Rung: 35 %
SOR LBL Q19:8 RET EOR
% Rung: 36 %
SOR END EOR

LADDER 20
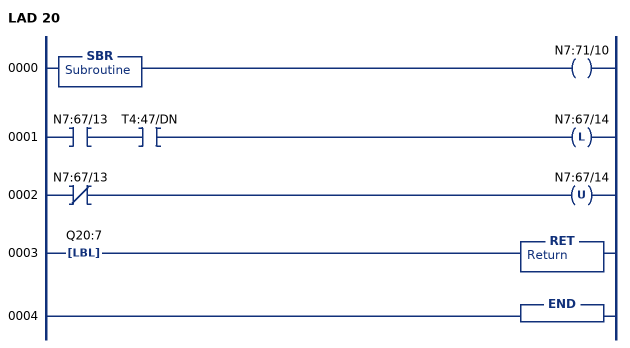
% Rung: 0 %
SOR SBR OTE N7:71/10 EOR
% Rung: 1 %
SOR XIC N7:67/13 XIC T4:47/DN OTL N7:67/14 EOR
% Rung: 2 %
SOR XIO N7:67/13 OTU N7:67/14 EOR
% Rung: 3 %
SOR LBL Q20:7 RET EOR
% Rung: 4 %
SOR END EOR

LADDER 21
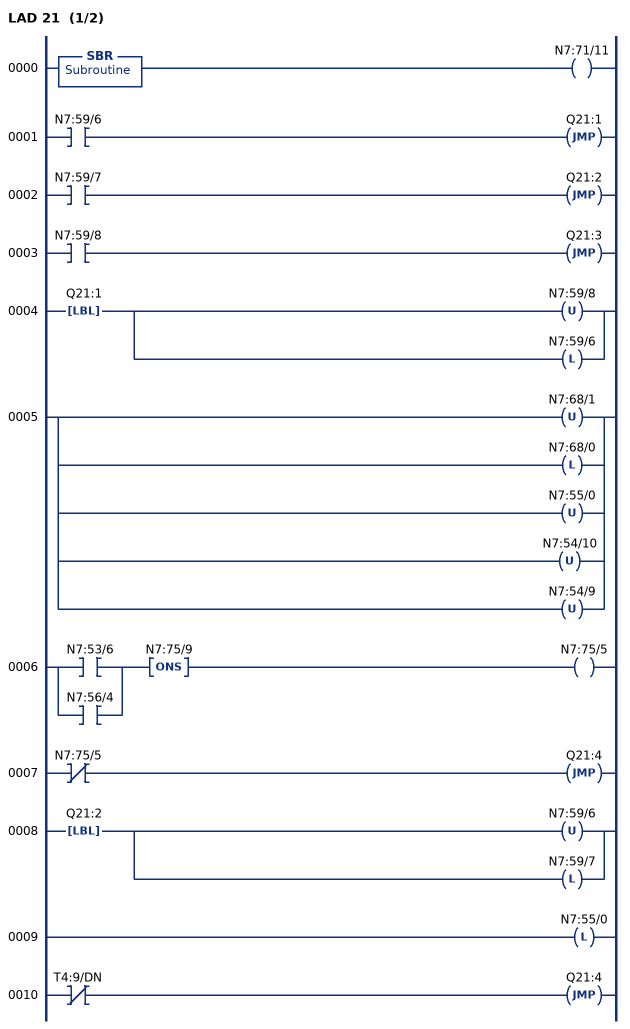
% Rung: 0 %
SOR SBR OTE N7:71/11 EOR
% Rung: 1 %
SOR XIC N7:59/6 JMP Q21:1 EOR
% Rung: 2 %
SOR XIC N7:59/7 JMP Q21:2 EOR
% Rung: 3 %
SOR XIC N7:59/8 JMP Q21:3 EOR
% Rung: 4 %
SOR LBL Q21:1 BST OTU N7:59/8 NXB OTL N7:59/6 BND EOR
% Rung: 5 %
SOR BST OTU N7:68/1 NXB OTL N7:68/0 NXB OTU N7:55/0 NXB OTU N7:54/10 NXB OTU N7:54/9 BND EOR
% Rung: 6 %
SOR BST XIC N7:53/6 NXB XIC N7:56/4 BND OSR N7:75/9 OTE N7:75/5 EOR
% Rung: 7 %
SOR XIO N7:75/5 JMP Q21:4 EOR
% Rung: 8 %
SOR LBL Q21:2 BST OTU N7:59/6 NXB OTL N7:59/7 BND EOR
% Rung: 9 %
SOR OTL N7:55/0 EOR
% Rung: 10 %
SOR XIO T4:9/DN JMP Q21:4 EOR

